(* IEC 61131-3 sources: plc_generation_empirical_study/datasets/_archive/pre_native_plcverif_20260810/tasks/C06_E01_three_part_counter, 2 files *)

(* ---- interface.st ---- *)
FUNCTION_BLOCK C06_E01_three_part_counter
VAR_INPUT
    PartPulse : BOOL;
    Reset : BOOL;
END_VAR
VAR_OUTPUT
    Count : INT;
    Complete : BOOL;
END_VAR
END_FUNCTION_BLOCK

(* ---- reference.st ---- *)
FUNCTION_BLOCK C06_E01_three_part_counter
VAR_INPUT
    PartPulse : BOOL;
    Reset : BOOL;
END_VAR
VAR_OUTPUT
    Count : INT;
    Complete : BOOL;
END_VAR
VAR
    PrevPart : BOOL := FALSE;
END_VAR

IF Reset THEN
    Count := 0;
ELSIF PartPulse AND (NOT PrevPart) AND (Count < 3) THEN
    Count := Count + 1;
END_IF;
Complete := Count = 3;
PrevPart := PartPulse;

END_FUNCTION_BLOCK
